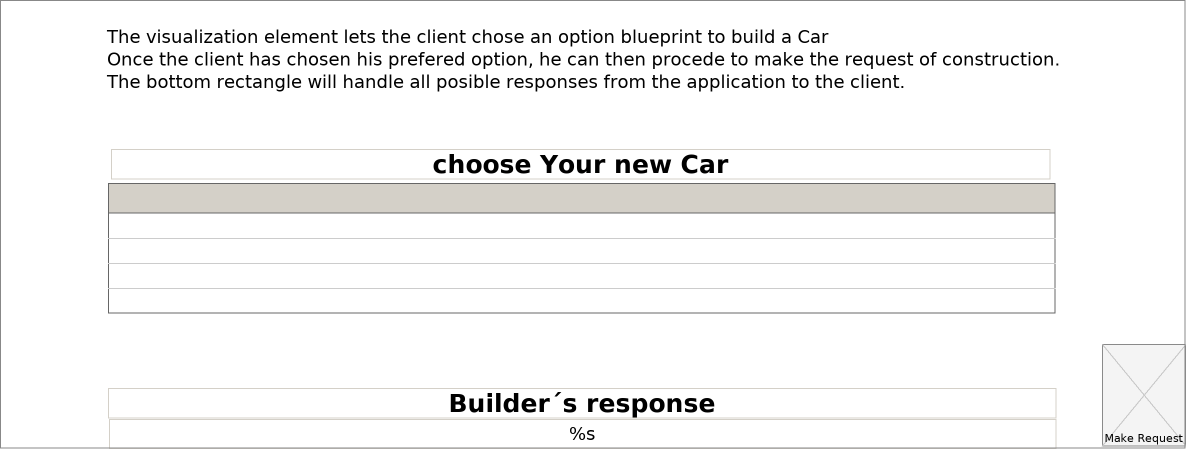
VISUALIZATION Visualization  // 1186x449
    Table (108,183 947x130), data array: MAIN.tableArray
        p3854506369: MAIN.tableArray[1,INDEX]
        p1892666644: MAIN.tableArray[2,INDEX]
        p338671338: MAIN.tableArray[3,INDEX]
        p2170511999: MAIN.tableArray[4,INDEX]
        p2232123230: Chassis Colour
        p511219082: Car type
        p1755163831: Motor dimensions
        p4092479075: Wheels type
        p1137915858: MAIN.iRow
        p1822360349: MAIN.bRow
    Textfield (111,149 939x30), "choose Your new Car"
    Textfield (108,388 948x30), "Builder´s response"
    Textfield (109,419 947x30), "%s", text variable: MAIN.sMessageLog
    Image (1102,344 84x102), "Make Request", image: VisuSymbols.Symbols.OK
        OnMouseClick: toggle MAIN.bRequest
    Label (104,10 953x99), "The visualization element lets the client chose an option blueprint to build a Car Once the client has chosen his prefered option, he can then procede to make the request of construction. The bottom rectangle will handle all posible responses from the application to the client."
END_VISUALIZATION

(* stored: Version 1.1.0.1, ProductVersion 3.1.4024.12
   Visu Visualization: Id {e5306a25-f821-4402-ba43-185485dda6c2} *)
